# EPICS autosave request: iocBoot/ioc6bmb/Galil_settings.req
file "CARS_24_motor_settings.req",     P=$(P)
file "galil_8_motor_extras.req",       P=$(P)Galil1:, M1=m1,  M2=m2,  M3=m3,  M4=m4,  M5=m5,  M6=m6,  M7=m7,  M8=m8
file "galil_8_motor_extras.req",       P=$(P)Galil2:, M1=m9,  M2=m10, M3=m11, M4=m12, M5=m13, M6=m14, M7=m15, M8=m16
file "galil_8_motor_extras.req",       P=$(P)Galil3:, M1=m18, M2=m19, M3=m20, M4=m21, M5=m22, M6=m23, M7=m23, M8=m24
